PROGRAM MAIN
VAR
	plc_fb:PLC_FB;
END_VAR

plc_fb
(
	//功能块输入参数
	PlcDataAll:=GVL.GvlDataAll,
    //功能块输出参数
	PlcBuffer=>Gvl.GvlBuffer,
	IndexBuffer=>Gvl.GvlIndexBuffer,
	
	// === 交互部分 ===
    Cmd_FeedRate     := GVL.Gvl_Cmd_FeedRate_Set,
    Cmd_SpindleSpeed := GVL.Gvl_Cmd_Spindle_Set,
    
    // 【新增】绑定上位机使能信号
    Cmd_Enable       := GVL.Gvl_Cmd_Enable_Override, 
    
    Act_FeedRate     => GVL.Gvl_Act_FeedRate_Real,
    
    // === 硬件IO部分 ===
    RawFeedRead_Gray     := GVL.Gvl_EL1018_FeedRead_Gray,
    OutFeedWrite_Gray    => GVL.Gvl_EL2008_FeedWrite_Gray,
    OutSpindleWrite_Gray => GVL.Gvl_EL2008_SpindleWrite_Gray,
    
    // 【修改】硬件有效位现在由 FB 的逻辑决定
    OutOverrideValid     => GVL.Gvl_Override_Valid

);

END_PROGRAM

(* stored: Version 1.1.0.1, ProductVersion 3.1.4024.12
   POU MAIN: Id {db0c4132-3096-48dc-8c70-9b713eb4aa34}, SpecialFunc None *)
